// TIA Portal V20 export
// export: Created 2025-12-01T14:57:05.6369738Z, ExportSetting None, DisplayName Totally Integrated Automation Portal, DisplayVersion V20 Update 3, DisplayName TIA Portal Openness, DisplayVersion V20 Update 3, DisplayName TIA Portal Version Control Interface, DisplayVersion V20 Update 3, DisplayName STEP 7 Professional, DisplayVersion V20 Update 3, DisplayName STEP 7 Safety, DisplayVersion V20 Update 2, DisplayName WinCC Basic/Comfort/Advanced, DisplayVersion V20 Update 3, DisplayName WinCC Professional, DisplayVersion V20 Update 3, DisplayName WinCC Unified, DisplayVersion V20 Update 3
FUNCTION "FC872_VerificarRutaEnMesa" : Void   // FC872, LAD
TITLE = Verificar Ruta de las UT's En la Mesa
{ S7_Optimized_Access := 'FALSE' }
AUTHOR : TRACKING
NAME : 20130301
VERSION : 3.1
// stored: AutoNumber false, SetENOAutomatically false
   VAR_INPUT
      Mesa : UInt;   // Numero de Mesa a Verificar
      TestGrupo : Bool;   // Si tiene que testear el Grupo
   END_VAR
   VAR_OUTPUT
      RutaOK : Bool;   // Todas las UT's tienen Ruta
   END_VAR
   VAR_TEMP
      MesaActual : UInt;
      NumeroUT : UInt;
      GrupoUT : UInt;
      Relleno : Byte;
      ValorReturn : Int;
   END_VAR
BEGIN

NETWORK
TITLE = Inicializar
// - Variables internas
// - Numero de DB que se necesitan
////////////////////////////////////////////////////////////////////////////
// --- Reseteo de las Variables

      SET;
      L     0;
      T     #GrupoUT;  // Grupo Desactivado
      R     #RutaOK;  // Salida Ruta NOK



NETWORK
TITLE = Bucle de la Cola de la Mesa
// Recorrer la Cola de Mesa, verificando las UT's:
//   + Bien si tienen todas ruta
//   + Bien que el grupo tienen todas ruta
////////////////////////////////////////////////////////////////////////////
// --- Recoger la Primera UT de la Mesa

      L     "DB810_ColasMesas".Colas[#Mesa].UT_PrimeraMesa;
      T     #NumeroUT;

      L     #NumeroUT;
      L     0;
      ==I;
      JC    Ruta_OK;  // - Hay Alguna UT en la Mesa ?

      L     "DB812_UTs_Control".UT[#NumeroUT].MesaActual;  // - Guardo la Mesa Actual
      T     #MesaActual;
      L     "DB812_UTs_Control".UT[#NumeroUT].Grupo;  // - Guardo el Grupo
      T     #GrupoUT;


////////////////////////////////////////////////////////////////////////////
// --- Comprobar que la Primera UT de la Mesa tiene Destino

      L     "DB812_UTs_Control".UT[#NumeroUT].MesaDestino;
      L     #MesaActual;
      ==I;
      JC    Ruta_NOK;  // Tiene Destino ?

      L     "DB812_UTs_Control".UT[#NumeroUT].MesaDestino;
      L     0;
      ==I;
      JC    Ruta_NOK;  // Tiene Destino ?


////////////////////////////////////////////////////////////////////////////
// --- Recorrer todas las UT's restantes de la Mesa
InicioBucleMesa:NOP   0;
      L     "DB812_UTs_Control".UT[#NumeroUT].UT_SiguienteMesa;
      T     #NumeroUT;

      L     #NumeroUT;
      L     0;
      ==I;
      JC    Ruta_OK;  // - Hay Alguna UT más ?

////////////////////////////////////////////////////////////////
// --- Testeo Si se Testea solo las UT's del Mismo Grupo

      AN    #TestGrupo;
      JC    SinTestearGrupo;  // Hay que testear Grupo ?

// --- Existe Grupo
      SET;
      L     #GrupoUT;
      L     0;
      ==I;
      JC    Ruta_NOK;

      SET;
      L     "DB812_UTs_Control".UT[#NumeroUT].Grupo;
      L     0;
      ==I;
      JC    Ruta_NOK;

// --- Comprobar Grupo
      SET;
      L     #GrupoUT;
      L     "DB812_UTs_Control".UT[#NumeroUT].Grupo;
      <>I;
      JC    Ruta_OK;  // Es del grupo a testear ?

SinTestearGrupo:NOP   0;


////////////////////////////////////////////////////////////////
// --- Comprobar Si tienen destino

      L     "DB812_UTs_Control".UT[#NumeroUT].MesaDestino;
      L     #MesaActual;
      ==I;
      JC    Ruta_NOK;  // Tiene Destino ?

      L     "DB812_UTs_Control".UT[#NumeroUT].MesaDestino;
      L     0;
      ==I;
      JC    Ruta_NOK;  // Tiene Destino ?

      JU    InicioBucleMesa;  // Continuar con la siguiente UT





NETWORK
TITLE = Respuesta
////////////////////////////////////////////////////////////////////////////
// --- Todas las UTs Tienen Destino

Ruta_OK:NOP   0;
      SET;
      S     #RutaOK;

      BE;


////////////////////////////////////////////////////////////////////////////
// --- No Todas las UTs Tienen Destino

Ruta_NOK:NOP   0;
      SET;
      R     #RutaOK;

      BE;



END_FUNCTION
